Staubli VAL3: TASK_MANAGER.pgx

program TASK_MANAGER()
begin
  while (bTaskManager)
    if taskStatus(sInputBuffering)==150
      taskKill(sInputBuffering)
      resetMotion()
      putln("Restart SIMPLE_MSG task.")
      taskCreate sInputBuffering,50,SIMPLE_MSG(trajMsg:prefix.nLength,trajMsg:header.nMsgType)
    endIf
  endWhile
end
